INTERFACE ITF_ControlElement_HMI_Init EXTENDS ITF_BaseControlElement, ITF_ControlElement_HMI_Connector

END_INTERFACE

(* stored: Version 1.1.0.1, ProductVersion 3.1.4024.15
   Itf ITF_ControlElement_HMI_Init: Id {a0e38302-8899-4b65-9b9b-3d94e0e55c99} *)
